// Interlock logic for the Amphos relay
FUNCTION F_AmphosEnable : BOOL
VAR_INPUT
	fAmphosVoltage : LREAL; // The Amphos voltage
	bEnabled : BOOL; // Whether the amphos enable signal is currently on
END_VAR
VAR_IN_OUT CONSTANT
	stAmphosSetpoints : ST_LaserSetpoints; // The Amphos setpoints
	stErrors : ST_ErrorStates; // Currently detected errors
END_VAR

IF stErrors.bHardwareFailure // Disable Amphos if there is a hardware failure
	OR stErrors.bAmphosBeam AND fAmphosVoltage < stAmphosSetpoints.nMinVoltage // Disable Amphos if there is a beam error
	OR stErrors.bAmphosBeam AND NOT bEnabled // Once amphos is disabled, keep it disabled until beam error is reset
THEN
	F_AmphosEnable := FALSE;
ELSE
	F_AmphosEnable := TRUE;
END_IF

END_FUNCTION

(* stored: Version 1.1.0.1, ProductVersion 3.1.4020.14
   POU F_AmphosEnable: Id {985578da-c888-4cd6-8fc2-8ee3835dc59d}, SpecialFunc None *)
